(*

.. <legal notes>

legal notes
=================
| SPDX-FileCopyrightText: © 2026 Oleksandr Tiutyk <trofimich@gmail.com>
| SPDX-License-Identifier: LGPL-3.0-only
| For details check: LGPL-3.0-only_

.. _LGPL-3.0-only: https://www.gnu.org/licenses/lgpl-3.0.en.html

.. </legal notes>

*)

INTERFACE IAutomationController EXTENDS Core.IExecutable, Automation.IAutomationComponent

{attribute 'monitoring' := 'call'}
PROPERTY DeviceCount : INT
GET
END_GET
END_PROPERTY

{attribute 'monitoring' := 'call'}
PROPERTY FINAL Diagnostics : REFERENCE TO AUTOMATION_CONTROLLER_DIAGNOSTICS
GET
END_GET
END_PROPERTY

PROPERTY ExceptionHandler : Core.IExceptionHandler
GET
END_GET
SET
END_SET
END_PROPERTY

METHOD FINAL Reset : BOOL
VAR_OUTPUT
	refuseReason : WSTRING(255);
END_VAR
END_METHOD

{attribute 'monitoring' := 'call'}
PROPERTY FINAL State : AUTOMATION_CONTROLLER_STATE
GET
END_GET
END_PROPERTY

{attribute 'monitoring' := 'call'}
PROPERTY FINAL StateChanged : BOOL
GET
END_GET
END_PROPERTY

{attribute 'monitoring' := 'call'}
PROPERTY StateName : STRING
GET
END_GET
END_PROPERTY

METHOD FINAL TryGetDeviceByIndex : Automation.IDevice
VAR_INPUT
	index : BYTE;
END_VAR
END_METHOD

END_INTERFACE

(* stored: Version 1.1.0.1
   Itf IAutomationController: Id {c1fb8ec2-f684-42e0-b4c9-67a265e32bf2}
   Property DeviceCount: Id {920b31c9-1e3d-40d6-8718-9c1ac02d1e5a}
   Get Get: Id {cfa98a1d-967c-4c63-aee3-493e072ad3fd}
   Property Diagnostics: Id {84c9e0c8-a36b-4d2d-aff4-16774b511646}
   Get Get: Id {4e9c458c-bb47-4a55-b6ab-f5871a54f704}
   Property ExceptionHandler: Id {a2483ac4-1f64-4cd4-b0d1-b3a7e19e7170}
   Get Get: Id {8c3a0814-e008-4f37-89bb-e6a536f3b087}
   Set Set: Id {9ba9462c-635a-4734-83f3-9cb6d147c579}
   Method Reset: Id {c67e1f83-8fec-4ed2-a85f-e7be08efc0f2}
   Property State: Id {0905c563-e105-4661-a19d-3580c163537e}
   Get Get: Id {7b01e8c1-82ac-4425-9e43-bb68fbd4a1e5}
   Property StateChanged: Id {e430642d-aaaf-4de3-a2b0-d4408db00024}
   Get Get: Id {43b05a9c-c420-416f-92ac-d40069def892}
   Property StateName: Id {e14367c7-04b5-4b25-ba36-2e091c6b443b}
   Get Get: Id {cc34a376-4466-4151-947c-23fbceb44621}
   Method TryGetDeviceByIndex: Id {c9989e47-fbd9-4c29-a256-afc552355c8f} *)
